(* IEC 61131-3 sources: crb-codesys/retrieval/output/codesys_repo/Decorator_Application/FUN, 22 files *)

(* ---- ConcreteComponment.st ---- *)
{attribute 'enable_dynamic_creation'}
//This class creates the most basic object well called. This object is to be decorated
FUNCTION_BLOCK ConcreteComponent IMPLEMENTS Component_Interface
VAR_INPUT
END_VAR
VAR_OUTPUT
END_VAR
VAR
	//String field to store the description of the object
	sDescription : STRING;
	//Real field to store the value of the object
	rValue : REAL;
END_VAR

(* ---- ConcreteDecoratorA.st ---- *)
 {attribute 'enable_dynamic_creation'}
//This class acts as a decorating class. It adds responsibilities and functionality to the component
FUNCTION_BLOCK ConcreteDecoratorA EXTENDS Decorator
VAR_INPUT
	//Reference to store the component to be decorated
	tempInputComponent : Component_Interface;
END_VAR
VAR_OUTPUT
END_VAR
VAR
END_VAR

(* ---- ConcreteDecoratorB.st ---- *)
{attribute 'enable_dynamic_creation'}
//This class acts as a decorating class. It adds responsibilities and functionality to the component
FUNCTION_BLOCK ConcreteDecoratorB EXTENDS Decorator
VAR_INPUT
	//Reference to store the component to be decorated
	tempInputComponent : Component_Interface;
END_VAR
VAR_OUTPUT
END_VAR
VAR
END_VAR

(* ---- ConcreteDecoratorC.st ---- *)
{attribute 'enable_dynamic_creation'}
//This class acts as a decorating class. It adds responsibilities and functionality to the component
FUNCTION_BLOCK ConcreteDecoratorC EXTENDS Decorator
VAR_INPUT
	//Reference to store the component to be decorated
	tempInputComponent : Component_Interface;
END_VAR
VAR_OUTPUT
END_VAR
VAR
END_VAR

(* ---- Decorator.st ---- *)
{attribute 'enable_dynamic_creation'}
//This class mainteins the reference to a ConcreteComponent object and works as an interface
// for its subclasses to decorate the ConcreteComponent
FUNCTION_BLOCK Decorator IMPLEMENTS Component_Interface
VAR_INPUT
END_VAR
VAR_OUTPUT
END_VAR
VAR
	//Variable to save the state of the concrete component to be decorated
	tempComponent : Component_Interface;
	//String variable to save the Description of the component
	sDescription : STRING;
	//Real variable to save the Value of the component
	rValue : REAL;
END_VAR

(* ---- Componment_Interface_getDescription.st ---- *)
//Illustrative method of the pattern
METHOD getDescription : String
VAR_INPUT
END_VAR

(* ---- Componment_Interface_getValue.st ---- *)
//Ilustrative method of the pattern
METHOD getValue : REAL
VAR_INPUT
END_VAR

(* ---- ConcreteComponment_fb_init.st ---- *)
METHOD fb_init
VAR_INPUT
	//Needed values to instanciation
	bInitRetains : BOOL; // TRUE: the Retain-variables are initialized (reset warm / reset cold)
	bInCopyCode : BOOL;  // TRUE  the instance will be copied to the copy-code afterward (online change)
END_VAR
VAR
	//String field to store the description of the object
	sDescription : STRING;
	//Real field to store the value of the object
	rValue : REAL;
END_VAR

//Sets the default description for the objects of this class
THIS^.sDescription := 'Plain Component';
//Sets the default value for the objects of this class
THIS^.rValue := 4.0;

(* ---- ConcreteComponment_getDescription.st ---- *)
//Illustrative method of the pattern
METHOD getDescription : STRING
VAR_INPUT
END_VAR
VAR_OUTPUT
END_VAR
VAR
	//String field to store the description of the object
	sDescription : STRING;
	//Real field to store the value of the object
	rValue : REAL;
END_VAR

//Description of the plain object is given
getDescription := This^.sDescription;

(* ---- ConcreteComponment_getValue.st ---- *)
//Illustrative method of the pattern
METHOD getValue : REAL
VAR_INPUT
END_VAR
VAR_OUTPUT
END_VAR
VAR
	//String field to store the description of the object
	sDescription : STRING;
	//Real field to store the value of the object
	rValue : REAL;
END_VAR

//Assume we are going to calculate the cost os the object.
//The plain value (without extra decoration) is given
getValue := THIS^.rValue;

(* ---- ConcreteDecoratorA_fb_init.st ---- *)
//Constructor of the decorating class called at instanciation
METHOD fb_init
VAR_INPUT
	//Needed values to instanciation
	bInitRetains : BOOL; // TRUE: the Retain-variables are initialized (reset warm / reset cold)
	bInCopyCode : BOOL;  // TRUE  the instance will be copied to the copy-code afterward (online change)

	//Reference to the component to be decorated passed as input
	tempInputComponent : Component_Interface;
END_VAR

//Calls the constructor (fb_init) in its SUPER class (Decorator)
// in order to pass the component to be decorated to the Decorator constructor.
SUPER^.fb_init(TRUE, TRUE, tempInputComponent);
//Sets the default description for the objects of this class
THIS^.sDescription := ' Decorator A';
//Sets the default value for the objects of this class
THIS^.rValue := 0.5;

(* ---- ConcreteDecoratorA_getDescription.st ---- *)
//Illustrative method of the pattern
METHOD getDescription : STRING
VAR_INPUT
	//Reference to store the component to be decorated
	tempInputComponent : Component_Interface;
END_VAR

//Outputs the decorated description of the component by obtaining the description of the component
// to be decorated stored in tempComponet.getDescription() and then concatenates the decoration
// description( ' Decorator A' as example)
getDescription :=CONCAT(THIS^.tempComponent.getDescription() , THIS^.sDescription);

(* ---- ConcreteDecoratorA_getValue.st ---- *)
//Illustrative method of the pattern
METHOD getValue : REAL
VAR_INPUT
	//Reference to store the component to be decorated
	tempInputComponent : Component_Interface;
END_VAR

//Outputs the decorated cost of the component by obtaining the cost of the component to be decorated
// stored in tempComponent.getValue() and then adds the decoration value (0.5 as example)
getValue := tempComponent.getValue() + THIS^.rValue;

(* ---- ConcreteDecoratorB_fb_init.st ---- *)
//Constructor of the decorating class called at instanciation
METHOD fb_init
VAR_INPUT
	//Needed values to instanciation
	bInitRetains : BOOL; // TRUE: the Retain-variables are initialized (reset warm / reset cold)
	bInCopyCode : BOOL;  // TRUE  the instance will be copied to the copy-code afterward (online change)

	//Reference to the component to be decorated passed as input
	tempInputComponent : Component_Interface;
END_VAR

//Calls the constructor (fb_init) in its SUPER class (Decorator)
// in order to pass the component to be decorated to the Decorator constructor.
SUPER^.fb_init(TRUE, TRUE, tempInputComponent);
//Sets the default description for the objects of this class
THIS^.sDescription := ' Decorator B';
//Sets the default value for the objects of this class
THIS^.rValue := 0.35;

(* ---- ConcreteDecoratorB_getDescription.st ---- *)
//Illustrative method of the pattern
METHOD getDescription : STRING
VAR_INPUT
	//Reference to store the component to be decorated
	tempInputComponent : Component_Interface;
END_VAR
VAR_OUTPUT
END_VAR
VAR
END_VAR

//Outputs the decorated description of the component by obtaining the description of the component
// to be decorated stored in tempComponet.getDescription() and then concatenates the decoration
// description( ' Decorator B' as example)
getDescription :=CONCAT(THIS^.tempComponent.getDescription() , THIS^.sDescription);

(* ---- ConcreteDecoratorB_getValue.st ---- *)
//Illustrative method of the pattern
METHOD getValue : REAL
VAR_INPUT
	//Reference to store the component to be decorated
	tempInputComponent : Component_Interface;
END_VAR
VAR_OUTPUT
END_VAR
VAR
END_VAR

//Outputs the decorated cost of the component by obtaining the cost of the component to be decorated
// stored in tempComponent.getValue() and then adds the decoration value (0.35 as example)
getValue := tempComponent.getValue() + THIS^.rValue;

(* ---- ConcreteDecoratorC_fb_init.st ---- *)
//Constructor of the decorator class called at instanciation
METHOD fb_init
VAR_INPUT
	//Needed values to instanciation
	bInitRetains : BOOL; // TRUE: the Retain-variables are initialized (reset warm / reset cold)
	bInCopyCode : BOOL;  // TRUE  the instance will be copied to the copy-code afterward (online change)

	//Reference to the component to be decorated passed as input
	tempInputComponent : Component_Interface;
END_VAR

//Calls the constructor (fb_init) in its SUPER class (Decorator)
// in order to pass the component to be decorated to the Decorator constructor.
SUPER^.fb_init(TRUE, TRUE, tempInputComponent);
//Sets the default description for the objects of this class
THIS^.sDescription := ' Decorator C';
//Sets the default value for the objects of this class
THIS^.rValue := 0.15;

(* ---- ConcreteDecoratorC_getDescription.st ---- *)
(*Illustrative method of the pattern*)
METHOD getDescription : STRING
VAR_INPUT
	//Reference to store the component to be decorated
	tempInputComponent : Component_Interface;
END_VAR
VAR_OUTPUT
END_VAR
VAR
END_VAR

//Outputs the decorated description of the component by obtaining the description of the component
// to be decorated stored in tempComponet.getDescription() and then concatenates the decoration
// description( ' Decorator C' as example)
getDescription :=CONCAT(THIS^.tempComponent.getDescription() , THIS^.sDescription);

(* ---- ConcreteDecoratorC_getValue.st ---- *)
(*Ilustrative method of the pattern*)
METHOD getValue : REAL
VAR_INPUT
	//Reference to store the component to be decorated
	tempInputComponent : Component_Interface;
END_VAR
VAR_OUTPUT
END_VAR
VAR
END_VAR

//Outputs the decorated cost of the component by obtaining the cost of the component to be decorated
// stored in tempComponent.getValue() and then adds the decoration value (0.15 as example)
getValue := tempComponent.getValue() + THIS^.rValue;

(* ---- Decorator_fb_init.st ---- *)
//Constructor of the decorator class called at instanciation
METHOD fb_init
VAR_INPUT
	//Needed values to instanciation
	bInitRetains : BOOL; // TRUE: the Retain-variables are initialized (reset warm / reset cold)
	bInCopyCode : BOOL;  // TRUE  the instance will be copied to the copy-code afterward (online change)

	//Reference to the component to be decorated passed as input
	tempInputComponent : Component_Interface;
END_VAR

//This constructor stores the component to be decorated in its field tempComponent in orer to be used by all its subclasses
THIS^.tempComponent := tempInputComponent;

(* ---- Decorator_getDescription.st ---- *)
//Illustrative method of the pattern
METHOD getDescription : STRING
VAR_INPUT
END_VAR
VAR_OUTPUT
END_VAR
VAR
	//Variable to save the state of the concrete component to be decorated
	tempComponent : Component_Interface;
	//String variable to save the Description of the component
	sDescription : STRING;
	//Real variable to save the Value of the component
	rValue : REAL;
END_VAR

//Outputs the description of the component to be decorated tempComponent. If tempComponent is not an undecorated component (plain object)
// it means the program has to do at least 2 decorations. Then is going to output the previous decoration complete description
// to be used by the next decorator.
getDescription := THIS^.tempComponent.getDescription();

(* ---- Decorator_getValue.st ---- *)
//Illustrative method of the pattern
METHOD getValue : REAL
VAR_INPUT
END_VAR
VAR_OUTPUT
END_VAR
VAR
	//Variable to save the state of the concrete component to be decorated
	tempComponent : Component_Interface;
	//String variable to save the Description of the component
	sDescription : STRING;
	//Real variable to save the Value of the component
	rValue : REAL;
END_VAR

//Outputs the cost of the component to be decorated tempComponent. If tempComponent is not an undecorated component (plain object)
// it means the program has to do at least 2 decorations. Then is going to output the previous decoration complete value
// to be used by the next decorator.
getValue := tempComponent.getValue();
